(* LS Electric XG5000 project: LP531_SynchronizationExample *)
(* PLC LSPLC *)
(* module base 0 slot 0: Input/Output Module:XEM-DN/DP32HP (DC 24V Input, Transistor Output, 32 Contacts) *)
(* module base 0 slot 1: Internal Positioning:XBF-PO06E (Open Collector Type, 6 Axis) *)

PROGRAM XPM_SSSP_Example (* task: Scan Program *)
(* this program is an example of XPM_SSS *)
VAR
    Axis1_Move_FB : XPM_DST; (* fb to move axis 1 in this example *)
    Axis2_SSSP_FB : XPM_SSSP; (* axis 2 speed synchronization fb *)
    Direct_HomeFB1 : XPM_FLT; (* direct home fb for axis 1 *)
    Direct_HomeFB2 : XPM_FLT; (* direct home fb for axis 2 *)
    Estop_Axes : BOOL; (* command to estop axes. *)
    Estop_Axis1_FB : XPM_EMG; (* estop axis 1 *)
    Estop_Axis2_FB : XPM_EMG; (* estop axis 2 *)
    Home_Axes : BOOL; (* command to home axis 1 and axis 2. *)
    Reset_Axes : BOOL; (* command to reset error on axis 1 and axis2. *)
    Reset_Axis1_FB : XPM_RST; (* reset axis 1 error *)
    Reset_Axis2_FB : XPM_RST; (* reset axis 2 error *)
    Run_Example : BOOL; (* command to run the example.  Perform this after homing and reseting axis errors (if any are present) *)
END_VAR

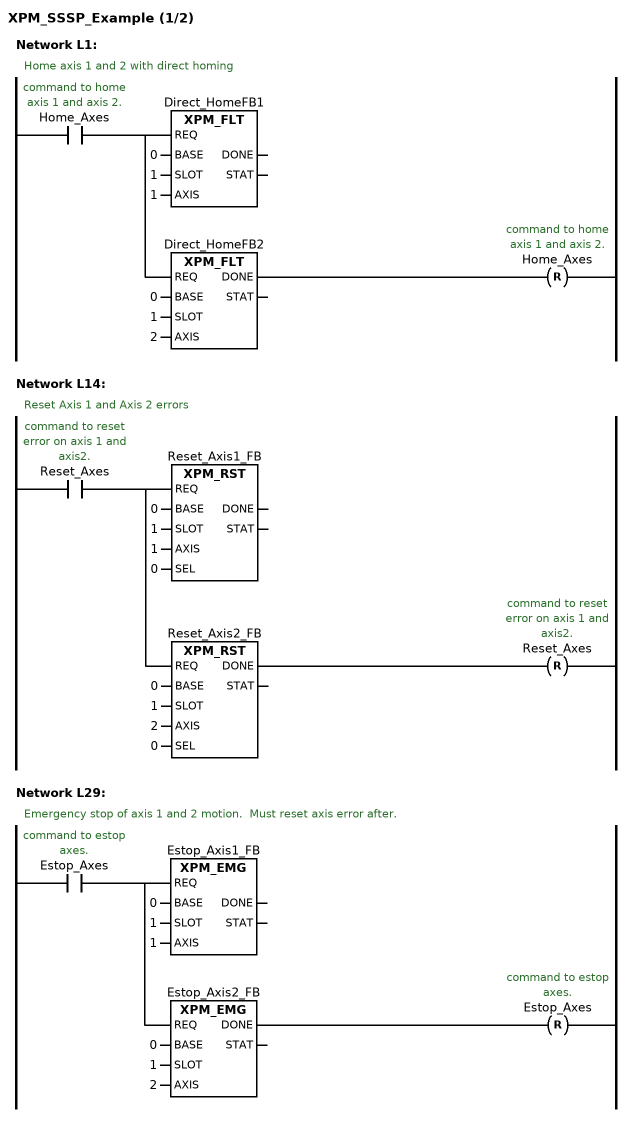
(* Home axis 1 and 2 with direct homing *)
(* Rung L1 *)
Direct_HomeFB1(REQ := Home_Axes, BASE := 0, SLOT := 1, AXIS := 1);
Direct_HomeFB2(REQ := Home_Axes, BASE := 0, SLOT := 1, AXIS := 2);
IF Direct_HomeFB2.DONE THEN Home_Axes := FALSE; END_IF;
(* Reset Axis 1 and Axis 2 errors *)
(* Rung L14 *)
Reset_Axis1_FB(REQ := Reset_Axes, BASE := 0, SLOT := 1, AXIS := 1, SEL := 0);
Reset_Axis2_FB(REQ := Reset_Axes, BASE := 0, SLOT := 1, AXIS := 2, SEL := 0);
IF Reset_Axis2_FB.DONE THEN Reset_Axes := FALSE; END_IF;
(* Emergency stop of axis 1 and 2 motion.  Must reset axis error after. *)
(* Rung L29 *)
Estop_Axis1_FB(REQ := Estop_Axes, BASE := 0, SLOT := 1, AXIS := 1);
Estop_Axis2_FB(REQ := Estop_Axes, BASE := 0, SLOT := 1, AXIS := 2);
IF Estop_Axis2_FB.DONE THEN Estop_Axes := FALSE; END_IF;

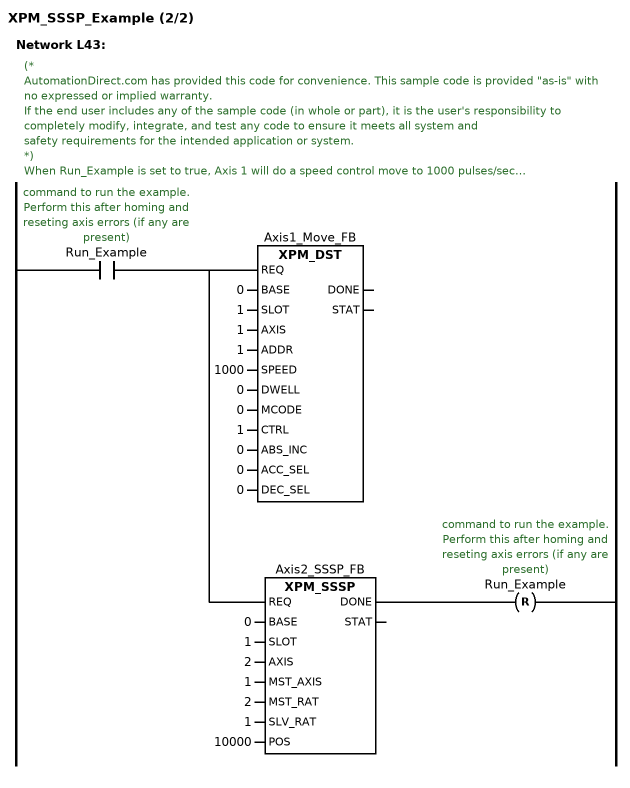
(* ( * / AutomationDirect.com has provided this code for convenience. This sample code is provided "as-is" with no expressed or implied warranty. / If the end user includes any of the sample code (in whole or part), it is the user's responsibility to completely modify, integrate, and test any code to ensure it meets all system and / safety requirements for the intended application or system. / * ) *)
(* When Run_Example is set to true, Axis 1 will do a speed control move to 1000 pulses/sec. / Axis 2 should synchronize speed at half the speed of Axis 1. *)
(* Rung L43 *)
Axis1_Move_FB(REQ := Run_Example, BASE := 0, SLOT := 1, AXIS := 1, ADDR := 1, SPEED := 1000, DWELL := 0, MCODE := 0, CTRL := 1, ABS_INC := 0, ACC_SEL := 0, DEC_SEL := 0);
Axis2_SSSP_FB(REQ := Run_Example, BASE := 0, SLOT := 1, AXIS := 2, MST_AXIS := 1, MST_RAT := 2, SLV_RAT := 1, POS := 10000);
IF Axis2_SSSP_FB.DONE THEN Run_Example := FALSE; END_IF;
END_PROGRAM

PROGRAM XPM_SSS_Example (* task: Scan Program *)
(* this program is an example of XPM_SSS *)
VAR
    Axis1_Move_FB : XPM_DST; (* fb to move axis 1 in this example *)
    Axis2_SSS_FB : XPM_SSS; (* axis 2 speed synchronization fb *)
    Direct_HomeFB1 : XPM_FLT; (* direct home fb for axis 1 *)
    Direct_HomeFB2 : XPM_FLT; (* direct home fb for axis 2 *)
    Estop_Axes : BOOL; (* command to estop axes. *)
    Estop_Axis1_FB : XPM_EMG; (* estop axis 1 *)
    Estop_Axis2_FB : XPM_EMG; (* estop axis 2 *)
    Home_Axes : BOOL; (* command to home axis 1 and axis 2. *)
    Reset_Axes : BOOL; (* command to reset error on axis 1 and axis2. *)
    Reset_Axis1_FB : XPM_RST; (* reset axis 1 error *)
    Reset_Axis2_FB : XPM_RST; (* reset axis 2 error *)
    Run_Example : BOOL; (* command to run the example.  Perform this after homing and reseting axis errors (if any are present) *)
END_VAR

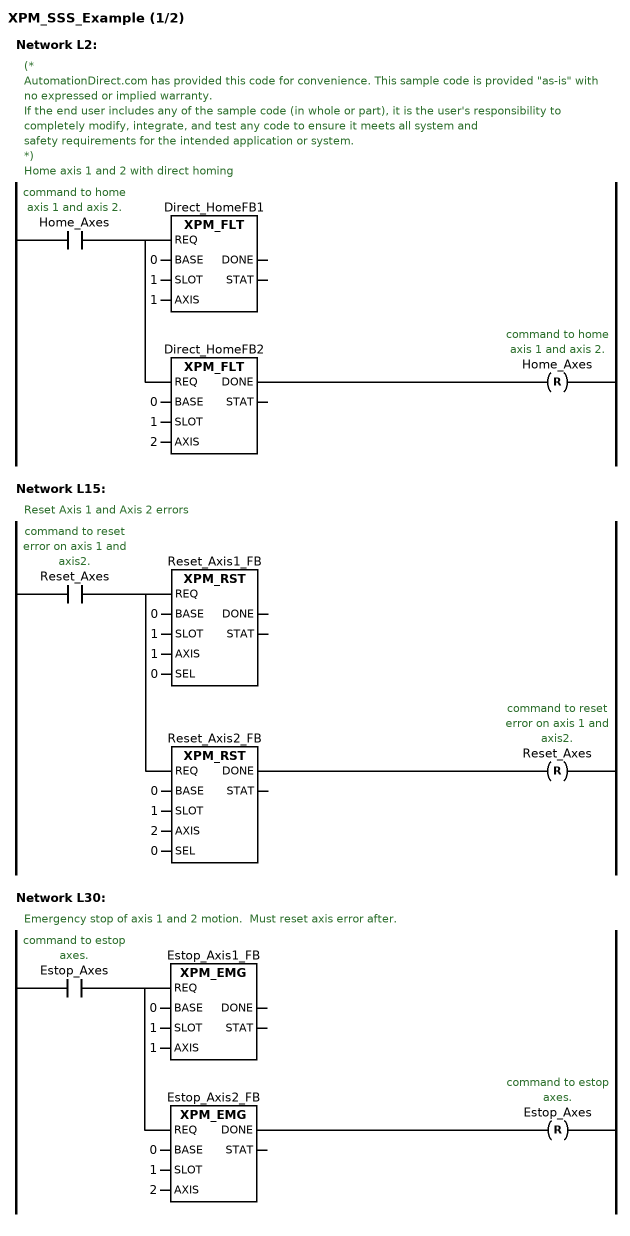
(* ( * / AutomationDirect.com has provided this code for convenience. This sample code is provided "as-is" with no expressed or implied warranty. / If the end user includes any of the sample code (in whole or part), it is the user's responsibility to completely modify, integrate, and test any code to ensure it meets all system and / safety requirements for the intended application or system. / * ) *)
(* Home axis 1 and 2 with direct homing *)
(* Rung L2 *)
Direct_HomeFB1(REQ := Home_Axes, BASE := 0, SLOT := 1, AXIS := 1);
Direct_HomeFB2(REQ := Home_Axes, BASE := 0, SLOT := 1, AXIS := 2);
IF Direct_HomeFB2.DONE THEN Home_Axes := FALSE; END_IF;
(* Reset Axis 1 and Axis 2 errors *)
(* Rung L15 *)
Reset_Axis1_FB(REQ := Reset_Axes, BASE := 0, SLOT := 1, AXIS := 1, SEL := 0);
Reset_Axis2_FB(REQ := Reset_Axes, BASE := 0, SLOT := 1, AXIS := 2, SEL := 0);
IF Reset_Axis2_FB.DONE THEN Reset_Axes := FALSE; END_IF;
(* Emergency stop of axis 1 and 2 motion.  Must reset axis error after. *)
(* Rung L30 *)
Estop_Axis1_FB(REQ := Estop_Axes, BASE := 0, SLOT := 1, AXIS := 1);
Estop_Axis2_FB(REQ := Estop_Axes, BASE := 0, SLOT := 1, AXIS := 2);
IF Estop_Axis2_FB.DONE THEN Estop_Axes := FALSE; END_IF;

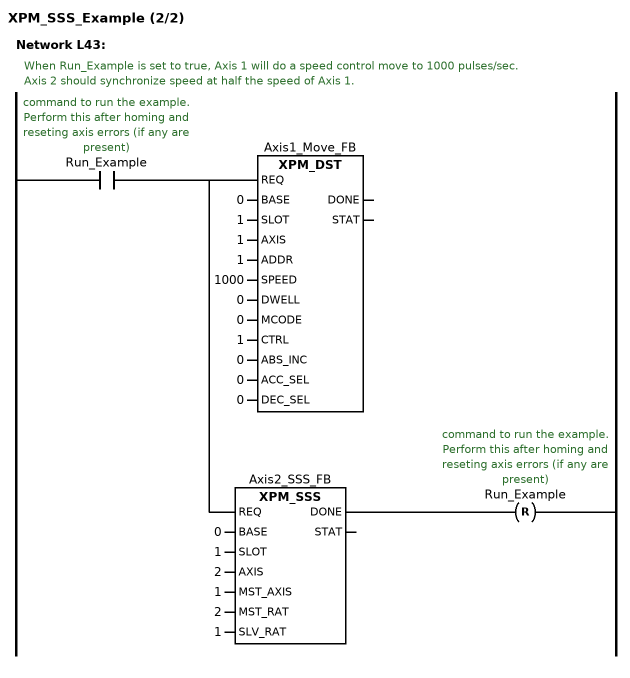
(* When Run_Example is set to true, Axis 1 will do a speed control move to 1000 pulses/sec. / Axis 2 should synchronize speed at half the speed of Axis 1. *)
(* Rung L43 *)
Axis1_Move_FB(REQ := Run_Example, BASE := 0, SLOT := 1, AXIS := 1, ADDR := 1, SPEED := 1000, DWELL := 0, MCODE := 0, CTRL := 1, ABS_INC := 0, ACC_SEL := 0, DEC_SEL := 0);
Axis2_SSS_FB(REQ := Run_Example, BASE := 0, SLOT := 1, AXIS := 2, MST_AXIS := 1, MST_RAT := 2, SLV_RAT := 1);
IF Axis2_SSS_FB.DONE THEN Run_Example := FALSE; END_IF;
END_PROGRAM

PROGRAM XPM_SSP_Example (* task: Scan Program *)
(* this program is an example of XPM_SSP *)
VAR
    Axis1_Move_FB : XPM_DST; (* fb to move axis 1 in this example *)
    Axis2_SSP_FB : XPM_SSP; (* axis 2 position synchronization fb *)
    Direct_HomeFB1 : XPM_FLT; (* direct home fb for axis 1 *)
    Direct_HomeFB2 : XPM_FLT; (* direct home fb for axis 2 *)
    Estop_Axes : BOOL; (* command to estop axes. *)
    Estop_Axis1_FB : XPM_EMG; (* estop axis 1 *)
    Estop_Axis2_FB : XPM_EMG; (* estop axis 2 *)
    Home_Axes : BOOL; (* command to home axis 1 and axis 2. *)
    Reset_Axes : BOOL; (* command to reset error on axis 1 and axis2. *)
    Reset_Axis1_FB : XPM_RST; (* reset axis 1 error *)
    Reset_Axis2_FB : XPM_RST; (* reset axis 2 error *)
    Run_Example : BOOL; (* command to run the example.  Perform this after homing and reseting axis errors (if any are present) *)
END_VAR

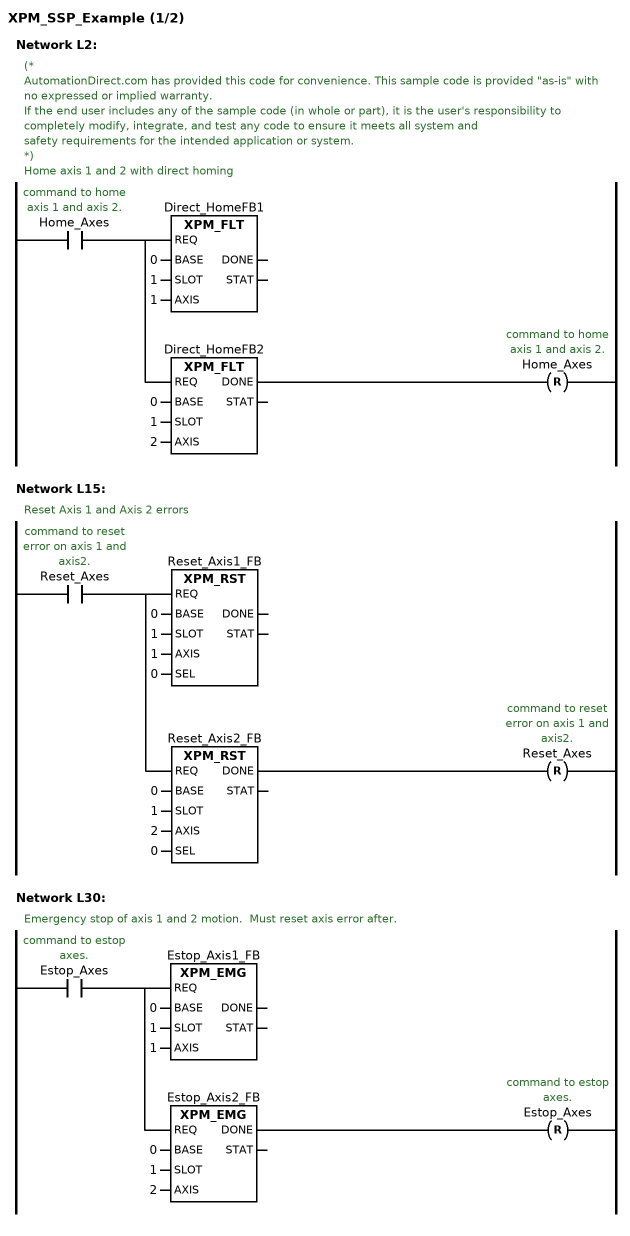
(* ( * / AutomationDirect.com has provided this code for convenience. This sample code is provided "as-is" with no expressed or implied warranty. / If the end user includes any of the sample code (in whole or part), it is the user's responsibility to completely modify, integrate, and test any code to ensure it meets all system and / safety requirements for the intended application or system. / * ) *)
(* Home axis 1 and 2 with direct homing *)
(* Rung L2 *)
Direct_HomeFB1(REQ := Home_Axes, BASE := 0, SLOT := 1, AXIS := 1);
Direct_HomeFB2(REQ := Home_Axes, BASE := 0, SLOT := 1, AXIS := 2);
IF Direct_HomeFB2.DONE THEN Home_Axes := FALSE; END_IF;
(* Reset Axis 1 and Axis 2 errors *)
(* Rung L15 *)
Reset_Axis1_FB(REQ := Reset_Axes, BASE := 0, SLOT := 1, AXIS := 1, SEL := 0);
Reset_Axis2_FB(REQ := Reset_Axes, BASE := 0, SLOT := 1, AXIS := 2, SEL := 0);
IF Reset_Axis2_FB.DONE THEN Reset_Axes := FALSE; END_IF;
(* Emergency stop of axis 1 and 2 motion.  Must reset axis error after. *)
(* Rung L30 *)
Estop_Axis1_FB(REQ := Estop_Axes, BASE := 0, SLOT := 1, AXIS := 1);
Estop_Axis2_FB(REQ := Estop_Axes, BASE := 0, SLOT := 1, AXIS := 2);
IF Estop_Axis2_FB.DONE THEN Estop_Axes := FALSE; END_IF;

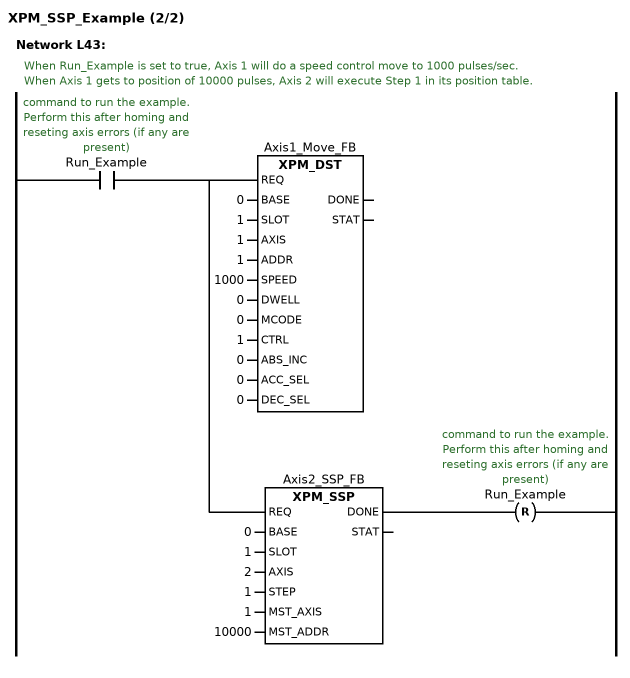
(* When Run_Example is set to true, Axis 1 will do a speed control move to 1000 pulses/sec. / When Axis 1 gets to position of 10000 pulses, Axis 2 will execute Step 1 in its position table. *)
(* Rung L43 *)
Axis1_Move_FB(REQ := Run_Example, BASE := 0, SLOT := 1, AXIS := 1, ADDR := 1, SPEED := 1000, DWELL := 0, MCODE := 0, CTRL := 1, ABS_INC := 0, ACC_SEL := 0, DEC_SEL := 0);
Axis2_SSP_FB(REQ := Run_Example, BASE := 0, SLOT := 1, AXIS := 2, STEP := 1, MST_AXIS := 1, MST_ADDR := 10000);
IF Axis2_SSP_FB.DONE THEN Run_Example := FALSE; END_IF;
END_PROGRAM